FUNCTION TryConvert_SINT_TO_USINT : BOOL
VAR_INPUT
	in : SINT;
	out : REFERENCE TO USINT;
END_VAR

IF in < DatatypeLimits.MIN_VALUE_OF_SINT_WHICH_CAN_BE_HELD_IN_A_USINT THEN
	RETURN;
END_IF

out := SINT_TO_USINT(in);
TryConvert_SINT_TO_USINT := TRUE;

END_FUNCTION

(* stored: Version 1.1.0.1, ProductVersion 3.1.4024.12
   POU TryConvert_SINT_TO_USINT: Id {d33d1894-8afa-439b-a953-747d240da659}, SpecialFunc None *)
